Fanuc KAREL source: kt00185.KL

-- PROVISIONAL review KL for V940-1; original PC SHA256 8e26c74208a2b973a9627c0134bed5b14ae332539369ae25ce8f49c4b1b44862
-- Incomplete behavior may be omitted. Consult companion uncertainty JSON. Do not deploy.
PROGRAM KT00185
%NOLOCKGROUP
VAR
  I2 : INTEGER
  OUT : INTEGER
-- UNRESOLVED_DECL H1 type=002017
BEGIN
  -- V9_ZERO_TABLE_METADATA_HINT layout=0001; no indexed target words; source/name/runtime held
  -- UNRESOLVED_PC offsets 5-19; opcodes 2E,22,9D,33,B4
  -- UNRESOLVED_PC offsets 24-35; opcodes 2E,23
  -- UNRESOLVED_PC offsets 40-62; opcodes 22,9D,33,B3,21,56,23
  -- UNRESOLVED_PC offsets 67-71; opcodes 7F
END KT00185
